# EPICS autosave request: cpscApp/Db/cpsc_axis_settings.req
$(P)$(M):Frequency.VAL
$(P)$(M):DriveFactor.VAL
$(P)$(M):StepSize.VAL
$(P)$(M):MovingDeadband.VAL
$(P)$(M):OpenLoopSteps.VAL
